FUNCTION_BLOCK PUBLIC CS_CodeTcp
VAR_INPUT
END_VAR
VAR_OUTPUT
END_VAR
VAR_IN_OUT
	
   iCode2:ICode;

END_VAR


VAR
	
	fbTcpCon:FB_SocketConnect;
	fbTcpSend:FB_SocketSend;
//	fbTcpSend2:FB_SocketSend;
	fbTcpRec:FB_SocketReceive;
	fbTcpClose: FB_SocketClose;
	bConnect: BOOL;
	bClose: BOOL;
	hTcpSock: T_HSOCKET;
	//aTcpSend:ARRAY[1..10] OF BYTE;
	//aTcpReceive:ARRAY[1..10] OF BYTE;	
	StrSend:STRING;
	StrReceive:STRING;
	fbUdpCreate:FB_SocketUdpCreate;
	hUdp: T_HSOCKET;
	bCreate: BOOL;
	port: UDINT:=60000;
	bSendTcp: BOOL;
	bReceiveTcp: BOOL;
	fbSwingHalt2: MC_Halt;
    TON01:TON;


	Lenth: UINT;
	StrSend2: STRING;
	bSendTcp2: BOOL;
	bCodeConError: BOOL;
	TON100:TON;
END_VAR




	Config();
	
	M_SendReceive();


	
	

	
	
	
	

	
	
	
	
	
	
	
	
	
	
	
	
	
	
	
	
	
(*	
   fbUdpCreate(
	sSrvNetId:= , 
	sLocalHost:= , 
	nLocalPort:= port, 
	bExecute:=bCreate , 
	tTimeout:= , 
	bBusy=> , 
	bError=> , 
	nErrId=> , 
	hSocket=> hUdp);
	
	
	*)

ACTION Config:



  IF iCode2.bComOpen THEN
	 bConnect:=TRUE;	
	 bClose:=FALSE;
	 iCode2.bComOpen:=FALSE;
  END_IF
  
   IF iCode2.bComClose THEN
	 bConnect:=FALSE;	
	 bClose:=TRUE;
	 iCode2.bComClose:=FALSE;
  END_IF 
  
  
  
fbTcpCon(
	sSrvNetId:= ''   ,          //       (*'169.254.46.193.1.1'*) , 
	sRemoteHost:='127.0.0.1'     , 
	nRemotePort:= port, 
	bExecute:=bConnect , 
	tTimeout:= , 
	bBusy=> , 
	bError=> , 
	nErrId=> , 
	hSocket=>hTcpSock );
	
fbTcpClose(
	sSrvNetId:= ''   , 
	hSocket:=hTcpSock , 
	bExecute:=bClose , 
	tTimeout:=T#5S , 
	bBusy=> , 
	bError=> , 
	nErrId=> );

IF fbTcpCon.bBusy THEN
	bConnect:=FALSE;
END_IF

IF fbTcpClose.bBusy THEN
   bClose:=FALSE;
END_IF
END_ACTION

ACTION M_SendReceive:

TON100(IN:= , PT:=T#12S , Q=> , ET=> );
  IF iCode2.bLON THEN
     StrSend:='LON16$R$N';
	 bSendTcp:=TRUE;
	 iCode2.bLON:=FALSE;
	 iCode2.bDone:=FALSE;
	 iCode2.bError:=FALSE;
	 iCode2.strCode:='';
	 Lenth:=SIZEOF(StrSend);
	 TON100.IN:=TRUE;
	// iCode.bCodeConError:=FALSE;
  END_IF

  IF iCode2.bLOFF THEN
     StrSend:='LOFF$R$N';
	 bSendTcp:=TRUE;
	 iCode2.bLOFF:=FALSE;
	 iCode2.bDone:=FALSE;
	 iCode2.bError:=FALSE;
	 iCode2.strCode:='';
	 Lenth:=SIZEOF(StrSend2);
  END_IF


fbTcpSend(
		sSrvNetId:= , 
		hSocket:=hTcpSock , 
		cbLen:=SIZEOF(StrSend), 
		pSrc:= ADR(StrSend), 
		bExecute:= bSendTcp, 
		tTimeout:= T#2S , 
		bBusy=> , 
		bError=> , 
		nErrId=> );
	
	TON01(IN:= bSendTcp, PT:= T#500MS, Q=> , ET=> );	
	IF TON01.Q THEN
		bSendTcp:=FALSE;
	END_IF
	
	
bReceiveTcp:=NOT bReceiveTcp;
fbTcpRec(
	sSrvNetId:= , 
	hSocket:= hTcpSock, 
	cbLen:=SIZEOF(StrReceive) , 
	pDest:=ADR(StrReceive) , 
	bExecute:=bReceiveTcp , 
	tTimeout:= T#5S, 
	bBusy=> , 
	bError=> , 
	nErrId=> , 
	nRecBytes=> );


(*
//IF 	StrReceive='ERROR$R0843160C8$R' OR StrReceive= 'ERROR$R' OR StrReceive='ER,' OR StrReceive=  'ERROR$R0842000C4$R' THEN
IF StrReceive<>''THEN
	IF LEN(STR:=StrReceive )>=14 AND LEN(STR:=StrReceive )<=20 AND FIND(STR1:=StrReceive , STR2:='ERROR' )=0 THEN
	  iCode2.strCode:=StrReceive;
	  StrReceive:='';
	  iCode2.bDone:=TRUE;
	ELSIF FIND(STR1:=StrReceive , STR2:='ERROR' )<>0 THEN 
	  iCode2.strCode:=StrReceive;
	  StrReceive:='';
	  iCode2.bError:=TRUE;
	END_IF
END_IF
			

IF  TON100.Q THEN
   IF StrReceive='' THEN
     // iCode.bCodeConError:=TRUE;	
   END_IF
   TON100.IN:=FALSE;
END_IF

//iCode.bCodeConError;

*)
END_ACTION

END_FUNCTION_BLOCK

(* stored: Version 1.1.0.1, ProductVersion 3.1.4024.9
   POU CS_CodeTcp: Id {6c1ec581-262d-4442-bd5f-fcd9ca6ef4f7}, SpecialFunc None
   Action Config: Id {4f4cac2d-0015-45f0-ad27-0550d1845503}
   Action M_SendReceive: Id {6fcda719-e557-4228-82f2-0f11bee1f35e} *)
